{attribute 'GeneratedUsingTerminal: BK1150-0000-0016'}
{attribute addProperty BoxType "BK1150-0000-0016"}
{attribute addProperty Description ""}
{attribute addProperty Physics "YY"}
{attribute addProperty Id "InputsAT %I*Inputs_CC16D1F40OutputsAT %I*Outputs_D8BAB3B30WcStateAT %I*WcState_9091E0EB2InfoDataAT %I*InfoData_90184F0C16"}
{attribute addProperty CRC "2734468583"}
{attribute addProperty Size "18"}
TYPE BK1150_A2FCADE7 EXTENDS EtcSlaveBoxBase_77A0E4A7 :
STRUCT
	{attribute addProperty Name "Inputs"}
	Inputs : Inputs_CC16D1F4;
	{attribute addProperty Name "Outputs"}
	Outputs : Outputs_D8BAB3B3;
	{attribute addProperty Name "WcState"}
	WcState : WcState_9091E0EB;
	{attribute addProperty Name "InfoData"}
	InfoData : InfoData_90184F0C;
END_STRUCT
END_TYPE

(* stored: Version 1.2.0.0, ProductVersion 3.1.4024.11
   DUT BK1150_A2FCADE7: Id {5a12ab83-d8fc-45be-a1a7-53ffb87e6092} *)
